VISUALIZATION Visualisierung  // 2x2
END_VISUALIZATION

(* stored: Version 1.1.0.1, ProductVersion 3.1.4024.4
   Visu Visualisierung: Id {32750c6d-8f0c-4433-8a33-2d59fa66803b} *)
